{attribute 'OPC.UA.DA' := '1'}
{attribute 'OPC.UA.DA.StructuredType' := '1'}
TYPE MinPowerMsg :
STRUCT
	Id : EPowerIlluminationFlow;
	MinPower : LREAL;
END_STRUCT
END_TYPE

(* stored: Version 1.1.0.1, ProductVersion 3.1.4024.3
   DUT MinPowerMsg: Id {aae37c77-8faf-4f10-ae2e-6fc341dc6219} *)
